RoboDK station: dofbot_DX_6_axis_generic_final_V1.0.0.rdk

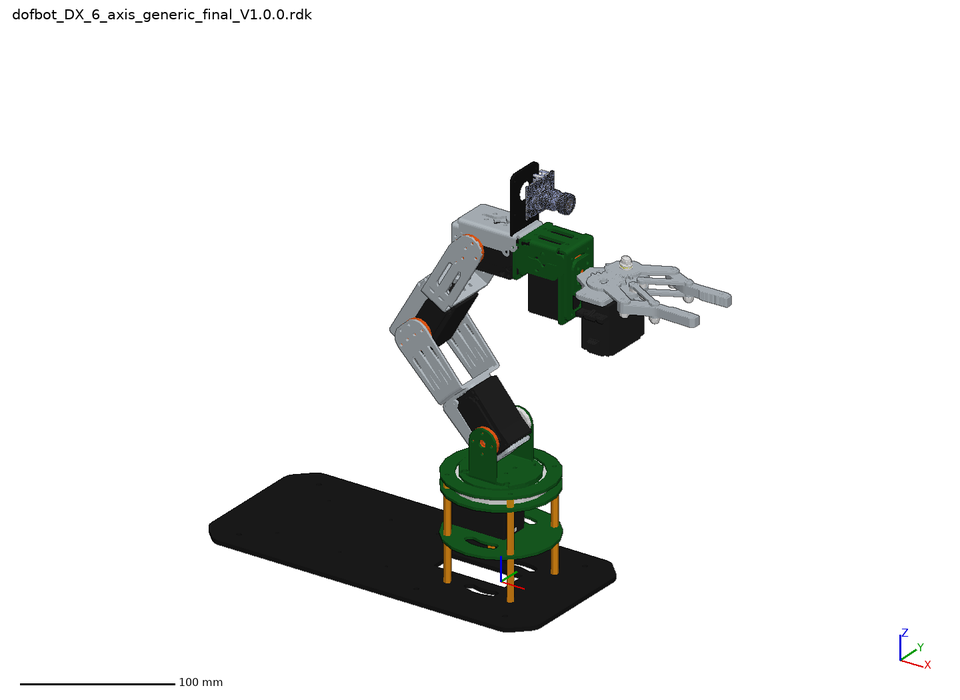
[picture v0: the station drawn from its stored meshes, robots at their saved joint values, targets as dots, program paths as lines]
Station dofbot_DX_6_axis_generic_final_V1.0.0 (saved by RoboDK 6.0.3). Poses are relative to the parent item; angles as X-Y-Z fixed-axis rotations.
  - frame Frame 1 at (0, 0, 0) mm
    - object dofbot_BASE_FRAME_add_axis at (0, 0, 0) mm, size 367.1 x 120 x 302.4 mm, geometry from dofbot_BASE_FRAME_add_axis.STEP
    - frame Frame 2 at (0, 0, 80) mm
      - object dofbot_LINK_1_add_axis at (0, 0, 0) mm, size 60.9 x 54.8 x 86.3 mm, geometry from dofbot_LINK_1_add_axis.STEP
        - frame Frame 3 at (0, 0, 27.5) mm, rotated rx -90 ry -50 rz 180 deg
          - object dofbot_LINK_2_add_axis at (0, 0, 0) mm, size 106.7 x 29.1 x 42.7 mm, geometry from dofbot_LINK_2_add_axis.STEP
          - frame Frame 4 at (82.85, 0, 0) mm, rotated rx 0 ry 0 rz -70 deg
            - object dofbot_LINK_3_add_axis at (0, 0, 0) mm, size 106.7 x 29.1 x 42.7 mm, geometry from dofbot_LINK_3_add_axis.STEP
            - frame Frame 5 at (82.85, 0, 0) mm, rotated rx 0 ry 0 rz -60 deg
              - object dofbot_LINK_4_add_axis at (0, 0, 0) mm, size 88 x 50 x 38.7 mm, geometry from dofbot_LINK_4_add_axis.STEP
              - frame Frame 6 at (70, -2.5, -1) mm, rotated rx 0 ry 90 rz 0 deg
                - object dofbot_LINK_5_add_axis at (0, 0, 0) mm, size 22.9 x 44 x 35.1 mm, geometry from dofbot_LINK_5_add_axis.STEP
                  - frame Frame 7 at (0, 0, 0) mm
                    - object dofbot_LINK_6_add_axis at (0, 0, 0) mm, size 62.7 x 55.3 x 110.3 mm, geometry from dofbot_LINK_6_add_axis.STEP
  - frame My Mechanism Base at (0, 1000, 0) mm
    - robot My Mechanism: 6 axes
        modified DH rows (alpha deg, a mm, theta deg, d mm): 0, 0, 0, 107.5; 90, 0, 130, 0; 0, 82.85, -70, 0; 0, 82.85, -60, 0; -90, 70, -90, 0; -90, 0, 0, 0
        joint limits [-200, -200, -200, -200, 0, -200] to [200, 200, 200, 200, 0, 200]; home [0, 0, 0, 0, 0, 0]; saved at [0, 0, 0, 0, 0, 0]
